// TIA Portal V17 export
// export: Created 2023-03-06T02:05:18.3692669Z, ExportSetting WithDefaults, DisplayName Totally Integrated Automation Portal, DisplayVersion V17 Update 4, DisplayName TIA Portal Openness, DisplayVersion V17 Update 4, DisplayName TIA Portal Version Control Interface, DisplayVersion V17, DisplayName STEP 7 Professional, DisplayVersion V17 Update 4, DisplayName STEP 7 Safety, DisplayVersion V17, DisplayName WinCC Professional, DisplayVersion V17 Update 4
DATA_BLOCK "LSNTP_Server_DB"   // DB123
VERSION : 2.1
// stored: AutoNumber false, DBAccessibleFromOPCUA true, DBAccessibleFromWebserver true, InstanceOfName LSNTP_Server, InstanceOfType FB
"LSNTP_Server"
   // VAR_INPUT
   //    init : Bool;
   //    referenceId : USInt;
   //    lastTimeSet : DTL;
   //    connID : CONN_OUC;
   //    hwID : HW_ANY;
   // END_VAR
   // VAR_OUTPUT
   //    error : Bool;
   //    statusID : Int;
   //    status : Word;
   // END_VAR
   // VAR
   //    InstTCON { S7_SetPoint := 'True'} : TCON;
   //    InstTURCV { S7_SetPoint := 'True'} : TURCV;
   //    InstTUSEND { S7_SetPoint := 'True'} : TUSEND;
   //    InstTDISCON { S7_SetPoint := 'True'} : TDISCON;
   //    statDiscon : Struct
   //       req : Bool;
   //       done : Bool;
   //       error : Bool;
   //       status : Word;
   //    END_STRUCT;
   //    statCon : Struct
   //       req : Bool;
   //       done : Bool;
   //       error : Bool;
   //       status : Word;
   //       param { S7_SetPoint := 'True'} : TCON_IP_v4;
   //    END_STRUCT;
   //    statRcv : Struct
   //       req : Bool;
   //       busy : Bool;
   //       error : Bool;
   //       ndr : Bool;
   //       len : UDInt;
   //       status : Word;
   //       addr { S7_SetPoint := 'True'} : TADDR_Param;
   //       tel { S7_SetPoint := 'True'} : "LSNTP_typeTelegram";
   //    END_STRUCT;
   //    statSend : Struct
   //       req : Bool;
   //       done : Bool;
   //       reqDone : Bool;
   //       error : Bool;
   //       status : Word;
   //       addr { S7_SetPoint := 'True'} : TADDR_Param;
   //       tel { S7_SetPoint := 'True'} : "LSNTP_typeTelegram";
   //    END_STRUCT;
   //    statState : Int;
   //    statEdge : Struct
   //       init : Bool;
   //    END_STRUCT;
   // END_VAR
BEGIN
END_DATA_BLOCK
